(* This function is for the MKS 722*)

FUNCTION_BLOCK FB_MKS722
VAR_IN_OUT
	
END_VAR
VAR_OUTPUT
	{attribute 'pytmc' := '
    pv: 
	'}
	VG	:	ST_VG;
END_VAR
VAR_INPUT
	i_rMinPressure	:	REAL;
	i_rMaxPressure	:	REAL;
END_VAR
VAR
	iTermBits: UINT := 32767 ; // The terminal's maximum value in bits
	rMinPressure: REAL;
	rVMin	:	REAL := 0.01; // Anything less than this voltage is considered disconnected
	rVMax :	REAL := 10.5; // Anything more than this is considered invalid
	rV	:REAL;
	
	(*IO*)
	i_iPRESS_R AT%I* :INT; // input Pressure // Link to analog Input
END_VAR



(* Real-value calculation *)
If (iTermBits=0) THEN iTermBits := 32767;END_IF
rV := 10*INT_TO_REAL(VG.i_iPRESS_R)/iTermBits;	


// Is the gauge plugged in, and within a reasonable range?
IF rV < rVMin THEN
	VG.eState := GaugeDisconnected;
ELSIF rV > rVMax THEN
	VG.eState := PressInvalid;
ELSIF VG.rPRESS >= rMinPressure AND VG.rPRESS <= i_rMaxPressure THEN
				VG.eState := Valid;
ELSIF VG.rPRESS < i_rMinPressure THEN
				VG.eState := ValidLo;
ELSE
				VG.eState := ValidHi;
END_IF
			
// Legacy Press OK boolean eval
VG.xPRESS_OK := VG.eState >= gc_GaugeValidState;

(*IO Soft Mapping*)
ACT_IO();

ACTION ACT_IO:
VG.i_iPRESS_R :=i_iPRESS_R;
END_ACTION

END_FUNCTION_BLOCK

(* stored: Version 1.1.0.1, ProductVersion 3.1.4024.3
   POU FB_MKS722: Id {367caa56-e444-4f21-b772-700d1462b7b8}, SpecialFunc None
   Action ACT_IO: Id {a9ca031f-8292-44da-bb18-9cf126ecf67e} *)
